FUNCTION_BLOCK FB_SV_Output
VAR_INPUT
	Stellung			: BOOL;
END_VAR
VAR_OUTPUT
	OUT_Stellung	: BOOL;
END_VAR
VAR
END_VAR

OUT_Stellung := Stellung;

END_FUNCTION_BLOCK

(* stored: Version 1.1.0.1, ProductVersion 3.1.4024.9
   POU FB_SV_Output: Id {e7b398e5-2eb1-4028-aa94-58f5fe50f259}, SpecialFunc None *)
